{attribute 'qualified_only'}
{attribute 'strict'}
TYPE E_AxisState :
(
	INIT := 0,
	READY,
	BUSY,
	ERROR
);
END_TYPE

(* stored: Version 1.1.0.1, ProductVersion 3.1.4020.12
   DUT E_AxisState: Id {0125a477-6e52-47e6-9aee-68f968d8bcaf} *)
